// TwinCAT 3 PLC project FunctionsPractice
// ProgramVersion: 3.1.4024.0
// libraries:
//   Tc2_ModbusSrv, * (Beckhoff Automation GmbH)
//   Tc2_Standard, * (Beckhoff Automation GmbH)
//   Tc2_System, * (Beckhoff Automation GmbH)
//   Tc3_Module, * (Beckhoff Automation GmbH)
// project tree:
//   / PlcTask.TcTTO
//   POUs/ FB_ModBusReadExample.TcPOU, FB_ModBusWriteExample.TcPOU, MAIN.TcPOU
// real-time tasks:
//   TASK PlcTask: cycle T#10ms, priority 20, ADS port 350
//   TASK PlcTask1: cycle T#10ms, priority 21, ADS port 351
//   TASK PlcTask2: cycle T#10ms, priority 22, ADS port 352

CONFIGURATION FunctionsPractice
    RESOURCE PLC ON TwinCAT3
        TASK PlcTask(INTERVAL := T#10ms, PRIORITY := 20);
        PROGRAM MAIN WITH PlcTask : MAIN;
    END_RESOURCE
END_CONFIGURATION

// ---- POUs/MAIN.TcPOU
PROGRAM MAIN
VAR
	fbRead : FB_ModBusReadExample;
	fbWrite : FB_ModBusWriteExample;
	
END_VAR

fbRead();
fbWrite();

END_PROGRAM

// ---- POUs/FB_ModBusReadExample.TcPOU
FUNCTION_BLOCK FB_ModBusReadExample

VAR
	fbReadCoil : FB_MBReadCoils;
	nReadValue : BYTE;
	fbTrig : R_TRIG;
	eState : (WAIT, TRIGGER, READ);
	nadsErrNumber : UDINT; 
	// Mapping a bit for a Coil (Address 0 in Modbus Poll)
    bMyCoil AT %MX0.0 : BOOL; 
    
    // Mapping a word for a Holding Register (Address 0 in Modbus Poll)
    nMyRegister AT %MB0 : WORD;
END_VAR

// 1. Always call the FB so it can process its internal state
fbReadCoil(
	sIPAddr    := '127.0.0.1', 
	nTCPPort   := 50502, 
	nUnitID    := 1, // Changed to 1, check your slave settings
	nQuantity  := 1, 
	nMBAddr    := 0, 
	cbLength   := SIZEOF(nReadValue), 
	pDestAddr  := ADR(nReadValue), 
	tTimeout   := T#5S
);

fbTrig();

CASE eState OF
	WAIT: 
		fbReadCoil.bExecute := FALSE; // Reset trigger for next time
		IF fbTrig.Q THEN
			eState := TRIGGER;
		END_IF
	
	TRIGGER:
		fbReadCoil.bExecute := TRUE; // Start the rising edge
		eState := READ;
		
	READ:
		IF NOT fbReadCoil.bBusy THEN
			IF fbReadCoil.bError THEN
				nadsErrNumber := fbReadCoil.nErrId;
			ELSE
				// Success! nReadValue now contains your data
				nadsErrNumber := 0;
			END_IF
			
			fbReadCoil.bExecute := FALSE; // Turn off the request
			eState := WAIT;
		END_IF
END_CASE

END_FUNCTION_BLOCK

// ---- POUs/FB_ModBusWriteExample.TcPOU
FUNCTION_BLOCK FB_ModBusWriteExample

VAR
	fbWriteCoil : FB_MBWriteSingleCoil;
	nWriteValue : WORD := 16#FF00;
	fbTrig : R_TRIG;
	eState : (WAIT, TRIGGER, WRITE);
	nadsErrNumber : UDINT; 
	// Mapping a bit for a Coil (Address 0 in Modbus Poll)
    bMyCoil AT %MX0.0 : BOOL; 
    
    // Mapping a word for a Holding Register (Address 0 in Modbus Poll)
    nMyRegister AT %MB0 : WORD;
END_VAR

// 1. Always call the FB so it can process its internal state
fbWriteCoil(
	sIPAddr:= '127.0.0.1' , 
	nTCPPort:= 50502, 
	nUnitID:= 1, 
	nMBAddr:= 0 , 
	nValue:= nWriteValue
	);
fbTrig();

CASE eState OF
	WAIT: 
		fbWriteCoil.bExecute := FALSE; // Reset trigger for next time
		IF fbTrig.Q THEN
			eState := TRIGGER;
		END_IF
	
	TRIGGER:
		fbWriteCoil.bExecute := TRUE; // Start the rising edge
		eState := WRITE;
		
	
	WRITE:
		IF NOT fbWriteCoil.bBusy THEN
			IF fbWriteCoil.bError THEN
				nadsErrNumber := fbWriteCoil.nErrId;
			ELSE
				// Success! nReadValue now contains your data
				nadsErrNumber := 0;
			END_IF
			
			fbWriteCoil.bExecute := FALSE; // Turn off the request
			eState := WAIT;
		END_IF
END_CASE

END_FUNCTION_BLOCK
